// SIMATIC STEP 7 (V5.x) project RLI-moteur
// CPU: CPU 315-2 PN/DP
// station: Matériel
// station: WC
// station: P_ADR_BUS
// program: Programme S7(1)

SYMBOL_TABLE
"capteur 1"	I 1.0	BOOL
"capteur 2"	I 1.1	BOOL
"sortie 1"	Q 1.0	BOOL
"sortie 2"	Q 1.1	BOOL
"VAT_1"	VAT 1	
END_SYMBOL_TABLE

ORGANIZATION_BLOCK OB 1
TITLE = "Main Program Sweep (Cycle)"
VERSION : 0.1
VAR_TEMP
  OB1_EV_CLASS : BYTE ;	//Bits 0-3 = 1 (Coming event), Bits 4-7 = 1 (Event class 1)
  OB1_SCAN_1 : BYTE ;	//1 (Cold restart scan 1 of OB 1), 3 (Scan 2-n of OB 1)
  OB1_PRIORITY : BYTE ;	//Priority of OB Execution
  OB1_OB_NUMBR : BYTE ;	//1 (Organization block 1, OB1)
  OB1_RESERVED_1 : BYTE ;	//Reserved for system
  OB1_RESERVED_2 : BYTE ;	//Reserved for system
  OB1_PREV_CYCLE : INT ;	//Cycle time of previous OB1 scan (milliseconds)
  OB1_MIN_CYCLE : INT ;	//Minimum cycle time of OB1 (milliseconds)
  OB1_MAX_CYCLE : INT ;	//Maximum cycle time of OB1 (milliseconds)
  OB1_DATE_TIME : DATE_AND_TIME ;	//Date and time OB1 started
END_VAR
BEGIN
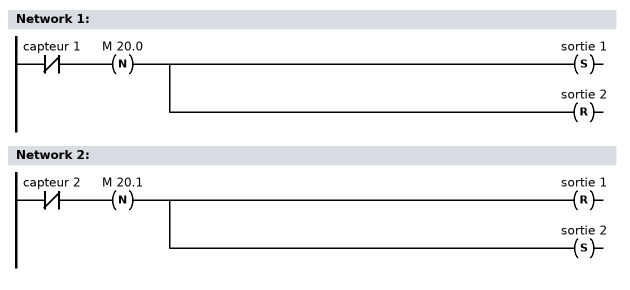
NETWORK
TITLE =
      AN    "capteur 1";
      FN    M 20.0;
      S     "sortie 1";
      R     "sortie 2";
NETWORK
TITLE =
      AN    "capteur 2";
      FN    M 20.1;
      R     "sortie 1";
      S     "sortie 2";
END_ORGANIZATION_BLOCK
